// TIA Portal V17 program export: 0 tag tables, 0 data types, 2 data blocks, 3 code blocks (in call order from the OBs), 0 instance data blocks

DATA_BLOCK "DB_ActivePopup"   // DB1
{ S7_Optimized_Access := 'TRUE' }
VERSION : 0.1
// stored: AutoNumber true, DBAccessibleFromOPCUA true, DBAccessibleFromWebserver true, IsOnlyStoredInLoadMemory false, IsRetainMemResEnabled false, IsWriteProtectedInAS false, MemoryReserve 100
   VAR
      Valve01 { S7_SetPoint := 'True'} : "UDT_ActivePopup";
      Heater01 { S7_SetPoint := 'True'} : "UDT_ActivePopup";
      Fan01 { S7_SetPoint := 'True'} : "UDT_ActivePopup";
   END_VAR
BEGIN
END_DATA_BLOCK

DATA_BLOCK "DB_Components"   // DB2
{ S7_Optimized_Access := 'TRUE' }
VERSION : 0.1
// stored: AutoNumber true, DBAccessibleFromOPCUA true, DBAccessibleFromWebserver true, IsOnlyStoredInLoadMemory false, IsRetainMemResEnabled false, IsWriteProtectedInAS false, MemoryReserve 100
   VAR
      Valve01 { S7_SetPoint := 'True'} : "UDT_ComponentPopup";   // 阀门
      Heater01 { S7_SetPoint := 'True'} : "UDT_ComponentPopup";   // 电加热
      Fan01 { S7_SetPoint := 'True'} : "UDT_ComponentPopup";   // 循环风机
   END_VAR
BEGIN
   Valve01.InfoTitle := '阀门01';
   Valve01.InfoMessage := '是否确认开启阀门01？';
   Heater01.InfoTitle := '电加热01';
   Heater01.InfoMessage := '是否确认开启电加热01？';
   Fan01.InfoTitle := '循环风机01';
   Fan01.InfoMessage := '是否确认开启循环风机01？';
END_DATA_BLOCK

ORGANIZATION_BLOCK "Main"   // OB1, SCL, ProgramCycle
TITLE = "Main Program Sweep (Cycle)"
{ S7_Optimized_Access := 'TRUE' }
VERSION : 0.1
// stored: AutoNumber true, IsIECCheckEnabled false, SetENOAutomatically false
   VAR_INPUT
      Initial_Call : Bool;   // Initial call of this OB
      Remanence : Bool;   // =True, if remanent data are available
   END_VAR
BEGIN
   "ZBRI-1_DB"();
END_ORGANIZATION_BLOCK

ORGANIZATION_BLOCK "Startup"   // OB100, SCL, Startup
TITLE = "Complete Restart"
{ S7_Optimized_Access := 'TRUE' }
VERSION : 0.1
// stored: AutoNumber true, IsIECCheckEnabled false, SetENOAutomatically false
   VAR_INPUT
      LostRetentive : Bool;   // True if retentive data are lost
      LostRTC : Bool;   // True if date and time are lost
   END_VAR
BEGIN
   // === 阀门01 配置 ===
   "DB_Components".Valve01.SwitchCnt := 2;
   "DB_Components".Valve01.RealCnt := 0;
   "DB_Components".Valve01.InfoCnt := 2;
   "DB_Components".Valve01.InfoTitle := '阀门01';
   "DB_Components".Valve01.InfoMessage := '是否确认开启阀门01？';

   // === 电加热01 配置 ===
   "DB_Components".Heater01.SwitchCnt := 1;
   "DB_Components".Heater01.RealCnt := 3;
   "DB_Components".Heater01.InfoCnt := 2;
   "DB_Components".Heater01.InfoTitle := '电加热01';
   "DB_Components".Heater01.InfoMessage := '是否确认开启电加热01？';

   // === 循环风机01 配置 ===
   "DB_Components".Fan01.SwitchCnt := 1;
   "DB_Components".Fan01.RealCnt := 2;
   "DB_Components".Fan01.InfoCnt := 2;
   "DB_Components".Fan01.InfoTitle := '循环风机01';
   "DB_Components".Fan01.InfoMessage := '是否确认开启循环风机01？';
END_ORGANIZATION_BLOCK

FUNCTION_BLOCK "HMI弹窗"   // FB1, SCL
{ S7_Optimized_Access := 'TRUE' }
VERSION : 0.1
// stored: AutoNumber true, IsIECCheckEnabled false, IsRetainMemResEnabled false, MemoryReserve 100, SetENOAutomatically false, UDAEnableTagReadback false
   VAR_INPUT
      DoubleClickTime : Time := T#800MS;
      CompID : Int;   // 部件唯一ID（>0）
   END_VAR
   VAR_IN_OUT
      Comp : "UDT_ComponentPopup";   // 单个部件
      Active : "UDT_ActivePopup";   // 全局激活区（共享）
   END_VAR
   VAR_TEMP
      R_Click : Bool;
      tNow : Time;
      tDiff : Time;
      i : Int;
   END_VAR
BEGIN
   // ========== 1. 上升沿检测 ==========
   #R_Click := #Comp.ClickTrig AND NOT #Comp.LastClick;
   #Comp.LastClick := #Comp.ClickTrig;

   #tNow := TIME_TCK();

   // ========== 2. 点击逻辑 ==========
   IF #R_Click THEN
       IF #Comp.ClickCount = 0 THEN
           // ===== 首次点击 → 打开弹窗，把部件数据复制到激活区 =====
           #Comp.ClickCount := 1;
           #Comp.FirstClickTime := #tNow;
           #Comp.Active := TRUE;

           #Active.ActiveID := #CompID;
           #Active.Visible := TRUE;
           #Active.Confirmed := FALSE;     // 清确认标志
           #Active.ConfirmBtn := FALSE;
           #Active.CancelBtn := FALSE;

           // 复制当前部件值 → 激活区（让HMI显示原值）
           FOR #i := 1 TO 8 DO
               #Active.Switch[#i] := #Comp.Switch[#i];
               #Active.RealValue[#i] := #Comp.RealValue[#i];
           END_FOR;
           #Active.InfoTitle := #Comp.InfoTitle;
           #Active.InfoMessage := #Comp.InfoMessage;
           #Active.InfoSpare1 := #Comp.InfoSpare1;
           #Active.InfoSpare2 := #Comp.InfoSpare2;

           // 设置可见性
           FOR #i := 1 TO 8 DO
               #Active.SwitchEnable[#i] := (#i <= #Comp.SwitchCnt);
               #Active.RealEnable[#i] := (#i <= #Comp.RealCnt);
           END_FOR;
           FOR #i := 1 TO 4 DO
               #Active.InfoEnable[#i] := (#i <= #Comp.InfoCnt);
           END_FOR;

       ELSE
           // ===== 双击窗口内再次点击 → 取消并隐藏（丢弃修改）=====
           #tDiff := #tNow - #Comp.FirstClickTime;
           IF #tDiff <= #DoubleClickTime THEN
               #Comp.Active := FALSE;
               #Comp.ClickCount := 0;
               #Active.Visible := FALSE;
               #Active.ActiveID := 0;
               FOR #i := 1 TO 8 DO
                   #Active.SwitchEnable[#i] := FALSE;
                   #Active.RealEnable[#i] := FALSE;
               END_FOR;
               FOR #i := 1 TO 4 DO
                   #Active.InfoEnable[#i] := FALSE;
               END_FOR;
               // ⚠ 不写回 Comp，丢弃HMI上的临时修改
           ELSE
               // 超时算新一轮首次点击
               #Comp.ClickCount := 1;
               #Comp.FirstClickTime := #tNow;
           END_IF;
       END_IF;
   END_IF;

   // ========== 3. 双击窗口超时清计数 ==========
   IF #Comp.ClickCount = 1 THEN
       IF (#tNow - #Comp.FirstClickTime) > #DoubleClickTime THEN
           #Comp.ClickCount := 0;
       END_IF;
   END_IF;

   // ========== 4. 当此部件激活时，处理确认/取消 ==========
   IF #Comp.Active AND (#Active.ActiveID = #CompID) THEN

       // ===== 确认按钮：把激活区的值提交到部件 =====
       IF #Active.ConfirmBtn THEN
           #Active.ConfirmBtn := FALSE;     // 自复位

           // ✅ 只在确认时写回部件
           FOR #i := 1 TO 8 DO
               #Comp.Switch[#i] := #Active.Switch[#i];
               #Comp.RealValue[#i] := #Active.RealValue[#i];
           END_FOR;

           #Active.Confirmed := TRUE;       // 给主程序判断用

           // 确认后关闭弹窗（按需保留/取消）
           #Active.Visible := FALSE;
           #Active.ActiveID := 0;
           #Comp.Active := FALSE;
           #Comp.ClickCount := 0;
           FOR #i := 1 TO 8 DO
               #Active.SwitchEnable[#i] := FALSE;
               #Active.RealEnable[#i] := FALSE;
           END_FOR;
           FOR #i := 1 TO 4 DO
               #Active.InfoEnable[#i] := FALSE;
           END_FOR;
       END_IF;

       // ===== 取消按钮：丢弃修改，关闭弹窗 =====
       IF #Active.CancelBtn THEN
           #Active.CancelBtn := FALSE;
           #Active.Visible := FALSE;
           #Active.ActiveID := 0;
           #Comp.Active := FALSE;
           #Comp.ClickCount := 0;
           FOR #i := 1 TO 8 DO
               #Active.SwitchEnable[#i] := FALSE;
               #Active.RealEnable[#i] := FALSE;
           END_FOR;
           FOR #i := 1 TO 4 DO
               #Active.InfoEnable[#i] := FALSE;
           END_FOR;
           // ⚠ 不写回 Comp
       END_IF;

   END_IF;
END_FUNCTION_BLOCK
